FUNCTION delay : bool
VAR_INPUT
	last_time : TIME;
	tempo : TIME;
END_VAR
VAR
END_VAR

IF TIME() - last_time >= tempo THEN 
	delay := TRUE ;
ELSE
	delay := FALSE;
END_IF

END_FUNCTION

(* stored: Version 1.1.0.1, ProductVersion 3.1.4024.11
   POU delay: Id {755ff08c-1583-4f14-bf33-0f1bb8dabb05}, SpecialFunc None *)
